INTERFACE I_RpcManager

METHOD PUBLIC TryHandleIncomingRequest : BOOL
VAR_INPUT
	Request : I_Request;
	Response : I_ServerResponse;
END_VAR
END_METHOD

END_INTERFACE

(* stored: Version 1.1.0.1, ProductVersion 3.1.4024.12
   Itf I_RpcManager: Id {d99fa72b-7fb1-42c3-97f3-801a898a58d4}
   Method TryHandleIncomingRequest: Id {11067e62-ee28-49db-a7c0-6ca545413550} *)
